# EPICS StreamDevice protocol: laudaRE2xx/lRE2xx_RS485.proto
##################################################
#
# Protocol File
#
# Protocol file for Lauda Ecoline Staredition RE2xx
# Diamond Light Source, Oct 2008
#
# NOTES:
#
#
#
##################################################

##################################################
# General Settings
##################################################

ReplyTimeout = 1000;

###################################################
# Get functions
###################################################

# /// Read water bath temperature
getTempA {
   ExtraInput = Ignore;
   out "\$1_IN_PV_00\r";
   in "\$1_IN_PV_00\r\$1_ %f\r";
}

# /// Read over temperature status
getStatusA {
   ExtraInput = Ignore;
   Separator = "";
   out "\$1_STAT\r";
   in "\$1_STAT\r\$1_%7d\r";
}

###################################################
# Set functions
###################################################

# /// Set the setpoint for water temperature (temperature must be specific format (up to 3 digits before decimal point and up to 2 digits after decimal point).
setTempA {
   out "\$1_OUT_SP_00_%.2f\r";
   in "\$1_OK\r";
}

#############################################################
# Generic protocol
############################################################

# /// Use this send any command and get back the response (max 39 chars).
genA {
    ExtraInput = Ignore;
    out "%s\r";
    in "%39c"
}
